(* CoDeSys 2.3 library: check.lib *)

(* POU CheckBounds, ST *)
FUNCTION CheckBounds : DINT
VAR_INPUT
	index, lower, upper: DINT;
END_VAR
VAR
END_VAR
IF index < lower THEN
	CheckBounds := lower;
ELSIF index > upper THEN
	CheckBounds := upper;
ELSE CheckBounds := index;
END_IF
END_FUNCTION

(* POU CheckDivByte, ST *)
FUNCTION CheckDivByte : BYTE
VAR_INPUT
	divisor: BYTE;
END_VAR
VAR
END_VAR
IF divisor = 0 THEN
	CheckDivByte := 1;
ELSE
	CheckDivByte := divisor;
END_IF
END_FUNCTION

(* POU CheckDivDWord, ST *)
FUNCTION CheckDivDWord : DWORD
VAR_INPUT
	divisor: DWORD;
END_VAR
VAR
END_VAR
IF divisor = 0 THEN
	CheckDivDWord := 1;
ELSE
	CheckDivDWord := divisor;
END_IF
END_FUNCTION

(* POU CheckDivReal, ST *)
FUNCTION CheckDivReal : REAL
VAR_INPUT
	divisor: REAL;
END_VAR
VAR
END_VAR
IF divisor = 0 THEN
	CheckDivReal := 1;
ELSE
	CheckDivReal := divisor;
END_IF
END_FUNCTION

(* POU CheckDivWord, ST *)
FUNCTION CheckDivWord : WORD
VAR_INPUT
	divisor: WORD;
END_VAR
VAR
END_VAR
IF divisor = 0 THEN
	CheckDivWord := 1;
ELSE
	CheckDivWord := divisor;
END_IF
END_FUNCTION

(* POU CheckRangeSigned, ST *)
FUNCTION CheckRangeSigned : DINT
VAR_INPUT
	value, lower, upper: DINT;
END_VAR
VAR
END_VAR
IF value < lower THEN
	CheckRangeSigned := lower;
ELSIF value > upper THEN
	CheckRangeSigned := upper;
ELSE
	CheckRangeSigned := value;
END_IF
END_FUNCTION
